FUNCTION_BLOCK SWITCHER2 (* Basic Function Block Type *)
  (* Standard: 61499-2 *)
  (* Version 0.3, 2009-09-15, JHC, Holobloc Inc, Changed transition priorities. *)
  (* Version 0.2, 2003-12-04, JHC, Rockwell Automation, Renamed for better indexing. *)
  (* Version 0.1, 2002-11-05, JHC, Rockwell Automation, Corrected missing ST element in Algorithm REQ. *)
  (* Version 0.0, 2000-05-30, JHC, Rockwell Automation *)
  (* Compiler header: package fb.rt.icaru; *)
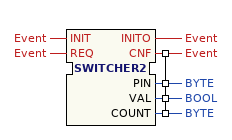
  EVENT_INPUT
    INIT; (* Initialization Request *)
    REQ; (* Normal Execution Request *)
  END_EVENT
  EVENT_OUTPUT
    INITO; (* Initialization Confirm *)
    CNF WITH PIN, VAL, COUNT; (* Execution Confirmation *)
  END_EVENT
  VAR_OUTPUT
    PIN : BYTE;
    VAL : BOOL;
    COUNT : BYTE;
  END_VAR
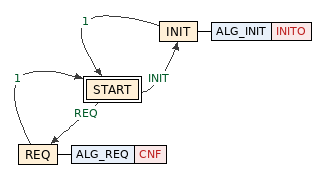
  EC_STATES
    START; (* Initial State *)
    INIT : ALG_INIT -> INITO; (* Initialization *)
    REQ : ALG_REQ -> CNF; (* Normal execution *)
  END_STATES
  EC_TRANSITIONS
    INIT TO START := 1;
    START TO REQ := REQ;
    START TO INIT := INIT;
    REQ TO START := 1;
  END_TRANSITIONS
  ALGORITHM ALG_INIT IN ST: (* Initialization algorithm *)
COUNT:=0;
VAL:=TRUE;
  END_ALGORITHM
  ALGORITHM ALG_REQ IN ST: (* Normally executed algorithm *)
COUNT := COUNT + 1;
 IF (COUNT > 3) THEN
   COUNT := 0;
   VAL := NOT VAL;
 END_IF;
 PIN := COUNT+26;
  END_ALGORITHM
END_FUNCTION_BLOCK
